// TIA Portal V17 export
// export: Created 2023-03-08T16:44:23.1874801Z, ExportSetting None, DisplayName Totally Integrated Automation Portal, DisplayVersion V17 Update 4, DisplayName TIA Portal Openness, DisplayVersion V17 Update 4, DisplayName TIA Portal Version Control Interface, DisplayVersion V17, DisplayName STEP 7 Professional, DisplayVersion V17 Update 4, DisplayName STEP 7 Safety, DisplayVersion V17, DisplayName WinCC Advanced / Unified PC, DisplayVersion V17 Update 4
DATA_BLOCK "DI"   // DB12
{ S7_Optimized_Access := 'TRUE' }
// stored: AutoNumber false, MemoryReserve 100
   VAR
      IR_READY : Bool;   // INGERSOL COMPRESSOR READY
      IR_TRIP : Bool;   // INGERSOL COMPRESSOR TRIP
      IR_LOADED : Bool;   // INGERSOL COMPRESSOR LOADED
      IR_AUTORESTART : Bool;   // INGERSOL COMPRESSOR AUTO STARTER
      IR_REMOTE : Bool;   // INGERSOL COMPRESSOR REMOTE
      AC_REMOTE : Bool;   // ATLAS COMPRESSOR REMOTE
      AC_RUNNING : Bool;   // ATLAS COMPRESSOR RUNNING
      AC_TRIP : Bool;   // ATLAS COMPRESSOR SHUTDOWN
      AC_READY : Bool;   // ATLAS COMPRESSOR PERMISSIVE TO START OK
      XA_001 : Bool;   // UCP HIGH INTERNAL TEMPERATURE
      XA_002 : Bool;   // UCP 24VDC POWER SUPPLY ALARM
      H1_SURGE_AL : Bool;   // HANWA 1 - SURGE ALARM
      H1_LS101_L : Bool;   // HANWA 1 - OIL LEVEL LOW ALARM
      H1_EM104_H : Bool;   // HANWA 1 - AOP TRIP ALARM
      H1_XV255_H : Bool;   // HANWA 1 - CHECK "DISCHARGE CHECK VALVE" ALARM
      H1_P_SG_AL : Bool;   // HANWA 1 - PRE SURGE ALARM
      H1_EH101_H : Bool;   // HANWA 1 - OIL HEATER TRIP ALARM
      H1_RTD_FAULT : Bool;   // HANWA 1 - RTD SIGNAL FAULT
      H1_AI_FAULT : Bool;   // HANWA 1 - ANALOG SIGNAL FAULT
      H1_SURGE_SD : Bool;   // HANWA 1 - SURGE DANGER
      H1_LS101_LL : Bool;   // HANWA 1 - OIL LEVEL VERY LOW DANGER
      H1_SP_FAULT : Bool;   // HANWA 1 - MOTOR START PANEL ON RESPONSE
      H1_AL_ON : Bool;   // HANWA 1 - GENERAL WARNING
      H1_SD_ON : Bool;   // HANWA 1 - GENERAL TRIP/FAULT
      H1_RE_ST_FAIL : Bool;   // HANWA 1 - REMOTE START FAILURE
      H1_RD_CSF : Bool;   // HANWA 1 - READY - CONTROLLER ERROR
      H2_SURGE_AL : Bool;   // HANWA 2 - SURGE ALARM
      H2_LS101_L : Bool;   // HANWA 2 - OIL LEVEL LOW ALARM
      H2_EM104_H : Bool;   // HANWA 2 - AOP TRIP ALARM
      H2_XV255_H : Bool;   // HANWA 2 - CHECK "DISCHARGE CHECK VALVE" ALARM
      H2_P_SG_AL : Bool;   // HANWA 2 - PRE SURGE ALARM
      H2_EH201_H : Bool;   // HANWA 2 - OIL HEATER TRIP ALARM
      H2_RTD_FAULT : Bool;   // HANWA 2 - RTD SIGNAL FAULT
      H2_AI_FAULT : Bool;   // HANWA 2 - ANALOG SIGNAL FAULT
      H2_SURGE_SD : Bool;   // HANWA 2 - SURGE DANGER
      H2_LS101_LL : Bool;   // HANWA 2 - OIL LEVEL VERY LOW DANGER
      H2_SP_FAULT : Bool;   // HANWA 2 - MOTOR START PANEL ON RESPONSE
      H2_AL_ON : Bool;   // HANWA 2 - GENERAL WARNING
      H2_SD_ON : Bool;   // HANWA 2 - GENERAL TRIP/FAULT
      H2_RE_ST_FAIL : Bool;   // HANWA 2 - REMOTE START FAILURE
      H2_RD_CSF : Bool;   // HANWA 2 - READY - CONTROLLER ERROR
   END_VAR
BEGIN
END_DATA_BLOCK
